TYPE _ST_HOME_ :
STRUCT
END_STRUCT
END_TYPE

(* stored: Version 1.1.0.1, ProductVersion 3.1.4022.18
   DUT _ST_HOME_: Id {f31c8671-26d7-48e1-8cc5-d112c10bd136} *)
